// TIA Portal V18 export
FUNCTION "SustainedOnOffHeating" : Void   // FC4, FBD
{ S7_Optimized_Access := 'TRUE' }
VERSION : 0.1
// stored: AutoNumber true, IsIECCheckEnabled false, SetENOAutomatically false, UDAEnableTagReadback false
   VAR_INPUT
      iUnitID : Int;
      cUpperState : Byte;
      rActual : Real;
      rSetPoint : Real;
      rHysteresis : Real;
      cRegulatorCfg : Byte;
   END_VAR
   VAR_OUTPUT
      cRegulatorState : Byte;
      cUnitStateTarget : Byte;
   END_VAR
BEGIN

REGION Network 1 (SCL)
   IF #rActual < #rSetPoint - #rHysteresis THEN
       #cUnitStateTarget := #cUpperState;
       #cRegulatorState := #cRegulatorCfg;
   ELSIF #cUnitStateTarget = #cUpperState AND #rActual > #rSetPoint + #rHysteresis THEN
       #cUnitStateTarget := 0;
       #cRegulatorState := 0;
   ELSE
       #cUnitStateTarget := 0;
       #cRegulatorState := 0;
   END_IF;
END_REGION
END_FUNCTION
